Fanuc KAREL source: kt00145.KL

-- PROVISIONAL review KL for V940-1; original PC SHA256 356e9b91f35d397bf8378046b9e5933ed05b0c78f4dc6aba716deca4fb9697d6
-- Incomplete behavior may be omitted. Consult companion uncertainty JSON. Do not deploy.
PROGRAM KT00145
%NOLOCKGROUP
VAR
  I2 : INTEGER
  OUT : INTEGER
-- UNRESOLVED_DECL Y1 type=002018
BEGIN
  -- V9_ZERO_TABLE_METADATA_HINT layout=0001; no indexed target words; source/name/runtime held
  -- UNRESOLVED_PC offsets 5-19; opcodes 2E,22,9D,33,B2
  -- UNRESOLVED_PC offsets 24-35; opcodes 2E,23
  -- UNRESOLVED_PC offsets 40-62; opcodes 22,9D,33,B1,21,55,23
  -- UNRESOLVED_PC offsets 67-71; opcodes 7F
END KT00145
